Fanuc TP program (LS listing): S103_PK_T20N50.LS

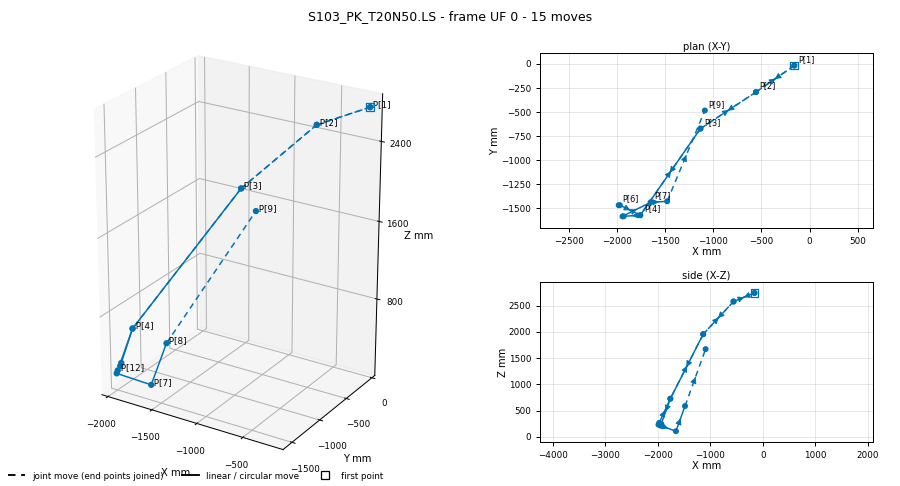
[picture p0: tool path of S103_PK_T20N50.LS in frame UF 0, 15 of 16 moves have a stored position in this frame; points joined in program order, loops and branches not executed]
/PROG  S103_PK_T20N50
/ATTR
OWNER		= MNEDITOR;
COMMENT		= "TL PCK TYP1 N50";
PROG_SIZE	= 4456;
CREATE		= DATE 19-12-16  TIME 15:28:32;
MODIFIED	= DATE 19-12-16  TIME 15:32:06;
FILE_NAME	= S103_PK_;
VERSION		= 0;
LINE_COUNT	= 161;
MEMORY_SIZE	= 4980;
PROTECT		= READ_WRITE;
STORAGE		= SHADOW;
TCD:  STACK_SIZE	= 0,
      TASK_PRIORITY	= 50,
      TIME_SLICE	= 0,
      BUSY_LAMP_OFF	= 0,
      ABORT_REQUEST	= 0,
      PAUSE_REQUEST	= 0;
DEFAULT_GROUP	= 1,*,*,*,*;
CONTROL_CODE	= 00000000 00000000;
/APPL
  HANDLING : TRUE ;
/MN
   1:  !******************************** ;
   2:  ! PATH - PK TOOL FROM N1=STA 70 ;
   3:  !******************************** ;
   4:  !* Robot ID: XXXXXR02B1 ;
   5:  !*    F-19XXXX ;
   6:  !* Line: XXXXXXXX ;
   7:  !* Platform: XX ;
   8:  !* Tool ID: TOOL xx ;
   9:  !* Program: S001_PK_TxxN3_R02 ;
  10:  !* Application: TOOL PICK ;
  11:  !******************************** ;
  12:  ! Author- Esys Automation ;
  13:  !******************************** ;
  14:   ;
  15:  !++++++++++++++++++++++++++++++++ ;
  16:  !ASSIGN PROGRAM PATH VALUES ;
  17:  !-------------------------------- ;
  18:  !Set ATI Tool and World UFrame ;
  19:  UTOOL_NUM=14 ;
  20:  UFRAME_NUM=0 ;
  21:  !++++++++++++++++++++++++++++++++ ;
  22:   ;
  23:  !******************************** ;
  24:  !BEGINNING OF PROGRAM PATH ;
  25:  !MOVE TO NEST 1 TOOL PICK ;
  26:  !******************************** ;
  27:   ;
  28:  !-------------------------------- ;
  29:  LBL[10:MOVE TO TL PICK] ;
  30:   ;
  31:  SET SEGMENT(52) ;
  32:  !SEG(52), Approach Tool Pick ;
  33:   ;
  34:J P[1] 100% CNT100    ;
  35:   ;
  36:J P[2] 100% CNT100    ;
  37:J P[3] 100% CNT100    ;
  38:   ;
  39:J P[4:Tool-Pick-Pounce] 100% CNT100    ;
  40:   ;
  41:L P[12] 500mm/sec CNT1    ;
  42:   ;
  43:L P[11] 30mm/sec FINE    ;
  44:   ;
  45:  !-------------------------------- ;
  46:  LBL[20:LATCH TOOL] ;
  47:  LATCH TOOL    ;
  48:   ;
  49:  !Add MH Ethernet Device from ;
  50:  !I/O Ethernet table ;
  51:  !which tool has ;
  52:   ;
  53:  !ADD DEVICE ONLINE CALLS ;
  54:  !WITHOUT STATUS CHECK ARG ;
  55:  !FOR ALL EOAT DEVICES ;
  56:  !CALL EN_ONLN(x,y) ;
  57:  !x = EOAT ENET Node # ;
  58:  !y = wait time ;
  59:  CALL EN_ONLN(31,5) ;
  60:  CALL EN_AROFF(31) ;
  61:   ;
  62:  !If TL LCH Pass, Return Home ;
  63:  !If TL LCH Fail, Unlatch TL, ;
  64:  !  MHFault, and Return Home ;
  65:  IF R[170]=1,JMP LBL[30] ;
  66:   ;
  67:  SELECT R[168]=6,JMP LBL[80] ;
  68:         ELSE,JMP LBL[99] ;
  69:   ;
  70:  !-------------------------------- ;
  71:  LBL[30:TOOL CHECK] ;
  72:   ;
  73:  ! Check if Tool Match with PLC ;
  74:  CALL TL_CHK_KM(R[156]) ;
  75:   ;
  76:  !If TL CHK Pass, Return Home ;
  77:  !If TL CHK Fail, Unlatch Tool, ;
  78:  !  MHFault, and Return Home ;
  79:  IF R[170]=1,JMP LBL[40] ;
  80:  IF R[170]=0,JMP LBL[905] ;
  81:   ;
  82:  !-------------------------------- ;
  83:  LBL[40:COMPLETE PATH] ;
  84:  !TL PK COMPLETE. MOVE AWAY ;
  85:  !AND RETURN HOME ;
  86:   ;
  87:  !Set New Tool and World Frame ;
  88:  UTOOL_NUM=2 ;
  89:  UFRAME_NUM=0 ;
  90:   ;
  91:  !Set Payload= Tool ;
  92:  R[221]=2    ;
  93:  PAYLOAD[R[221]] ;
  94:   ;
  95:  SET SEGMENT(53) ;
  96:  !SEG(53), Tool Pick Depart ;
  97:   ;
  98:L P[7] 100mm/sec FINE    ;
  99:   ;
 100:L P[8] 2000mm/sec CNT50    ;
 101:   ;
 102:J P[9] 100% CNT100    ;
 103:J P[10] 100% CNT100    ;
 104:   ;
 105:  ! Move To Home ;
 106:  JMP LBL[100] ;
 107:   ;
 108:  !-------------------------------- ;
 109:  LBL[80:LATCHING FAULT] ;
 110:  !MOVE BACK TO HOME WITHOUT TOOL ;
 111:  !on Reverse Path before Tool Pick ;
 112:   ;
 113:  UNLATCH TOOL    ;
 114:   ;
 115:  UFRAME_NUM=0 ;
 116:  UTOOL_NUM=14 ;
 117:   ;
 118:L P[6:PICK_T3_R1_N1] 50mm/sec FINE    ;
 119:   ;
 120:L P[5] 500mm/sec FINE    ;
 121:   ;
 122:L P[4:Tool-Pick-Pounce] 750mm/sec CNT100    ;
 123:   ;
 124:L P[3] 3000mm/sec CNT100    ;
 125:   ;
 126:J P[2] 100% CNT100    ;
 127:   ;
 128:J P[1] 100% CNT100    ;
 129:   ;
 130:  SET SEGMENT(63) ;
 131:  !SEG(63), Robot Move to Home ;
 132:   ;
 133:  R[132]=0    ;
 134:  GO[71]=0 ;
 135:   ;
 136:  ! Move To Home ;
 137:  JMP LBL[100] ;
 138:   ;
 139:  !-------------------------------- ;
 140:  LBL[99:ABORT PROGRAM] ;
 141:  MESSAGE[...] ;
 142:  MESSAGE[ABORT PROGRAM] ;
 143:  ABORT ;
 144:   ;
 145:  !-------------------------------- ;
 146:  LBL[100:END OF PROGRAM] ;
 147:  END ;
 148:   ;
 149:  !***********FAULTS*********** ;
 150:  LBL[905:Invalid Tool Num] ;
 151:  MESSAGE[...] ;
 152:  MESSAGE[TOOL CHANGER FAULT] ;
 153:  MESSAGE[ ROBOT LATCHED TO] ;
 154:  MESSAGE[ WRONG TOOL.] ;
 155:  MESSAGE[ GI[70] DOES NOT ] ;
 156:  MESSAGE[ MATCH TOOL ID ] ;
 157:  DO[523]=ON ;
 158:  UALM[3] ;
 159:  DO[523]=OFF ;
 160:  JMP LBL[80] ;
 161:   ;
/POS
P[1]{
   GP1:
	UF : 0, UT : 14,		CONFIG : 'N U B, 0, 0, 0',
	X =  -158.400  mm,	Y =   -15.894  mm,	Z =  2741.103  mm,
	W =   -91.792 deg,	P =     -.357 deg,	R =   122.600 deg
};
P[2]{
   GP1:
	UF : 0, UT : 14,		CONFIG : 'N U T, 0, 0, 0',
	X =  -557.806  mm,	Y =  -292.410  mm,	Z =  2577.899  mm,
	W =  -107.925 deg,	P =    -3.536 deg,	R =   122.979 deg
};
P[3]{
   GP1:
	UF : 0, UT : 14,		CONFIG : 'N U T, 0, 0, 0',
	X = -1134.710  mm,	Y =  -671.782  mm,	Z =  1955.941  mm,
	W =  -117.901 deg,	P =    -3.388 deg,	R =   113.635 deg
};
P[4:"Tool-Pick-Pounce"]{
   GP1:
	UF : 0, UT : 14,		CONFIG : 'N U T, 0, 0, 0',
	X = -1760.306  mm,	Y = -1572.902  mm,	Z =   727.655  mm,
	W =  -160.107 deg,	P =      .639 deg,	R =    91.877 deg
};
P[5]{
   GP1:
	UF : 0, UT : 14,		CONFIG : 'N U T, 0, 0, 0',
	X = -1972.818  mm,	Y = -1468.270  mm,	Z =   267.427  mm,
	W =  -160.182 deg,	P =     -.205 deg,	R =    91.920 deg
};
P[6:"PICK_T3_R1_N1"]{
   GP1:
	UF : 0, UT : 14,		CONFIG : 'N U T, 0, 0, 0',
	X = -1985.240  mm,	Y = -1468.564  mm,	Z =   232.950  mm,
	W =  -160.182 deg,	P =     -.205 deg,	R =    91.920 deg
};
P[7]{
   GP1:
	UF : 0, UT : 2,		CONFIG : 'N U T, 0, 0, 0',
	X = -1653.748  mm,	Y = -1439.220  mm,	Z =   109.203  mm,
	W =  -161.664 deg,	P =     1.002 deg,	R =    90.501 deg
};
P[8]{
   GP1:
	UF : 0, UT : 2,		CONFIG : 'N U T, 0, 0, 0',
	X = -1480.885  mm,	Y = -1428.210  mm,	Z =   587.612  mm,
	W =  -161.664 deg,	P =     1.002 deg,	R =    90.501 deg
};
P[9]{
   GP1:
	UF : 0, UT : 2,		CONFIG : 'N U T, 0, 0, 0',
	X = -1089.020  mm,	Y =  -483.560  mm,	Z =  1671.146  mm,
	W =  -119.401 deg,	P =    -2.194 deg,	R =   112.860 deg
};
P[10]{
   GP1:
	UF : 0, UT : 2,
	J1=  -145.477 deg,	J2=   -28.708 deg,	J3=    89.000 deg,
	J4=     2.573 deg,	J5=   -83.800 deg,	J6=   -90.000 deg
};
P[11]{
   GP1:
	UF : 0, UT : 14,		CONFIG : 'N U T, 0, 0, 0',
	X = -1945.725  mm,	Y = -1584.711  mm,	Z =   214.494  mm,
	W =  -160.107 deg,	P =      .639 deg,	R =    91.877 deg
};
P[12]{
   GP1:
	UF : 0, UT : 14,		CONFIG : 'N U T, 0, 0, 0',
	X = -1933.168  mm,	Y = -1583.913  mm,	Z =   249.246  mm,
	W =  -160.107 deg,	P =      .639 deg,	R =    91.877 deg
};
/END
